{attribute addProperty BoxType "EL3783-0000-0018"}
{attribute addProperty Id "U3_SamplesAT %I*ARRAY [0..19] OF INT32040"}
{attribute addProperty CRC "995984480"}
{attribute addProperty SizeInBites "320"}
{attribute addProperty SizeInBytes "40"}
TYPE L3_Voltage_Samples_3B5D8460 :
STRUCT
	{attribute addProperty Name "U3_Samples"}
	U3_Samples AT %I* : ARRAY [0..19] OF INT;
END_STRUCT
END_TYPE

(* stored: Version 1.2.0.0, ProductVersion 3.1.4024.9
   DUT L3_Voltage_Samples_3B5D8460: Id {55f49dcf-dda1-47a4-bb0b-5bd9d2d98374} *)
